FUNCTION_BLOCK FB_StationUnloadUc
VAR_INPUT
	Enable:				BOOL;
	System:				REFERENCE TO ST_System;
	Station:			REFERENCE TO ST_SystemStation;
	Error:				REFERENCE TO ST_Error;
	Setting:			REFERENCE TO ST_Setting;
	Recipe:				REFERENCE TO ST_Recipe;	
	Parameter:			REFERENCE TO ST_StationUnloadUc;
END_VAR
VAR_OUTPUT
END_VAR
VAR
	_i:					INT;
	_arrTon:		    ARRAY[0..20] OF TON;
	_arrFbErrorTag:		ARRAY[0..20] OF FB_ErrorTag;
	_arrState:			ARRAY[0..20] OF BOOL;
	_stHandshake: 		ST_StationUnloadUcHandshake;
END_VAR

A_Auto();
A_Home();

ACTION A_Auto:
CASE Station.iStepNow OF
	1000:
		Station.arrInfo[E_Language.Chinese]:="初始化完成 等待启动";
		IF Enable THEN
			Station.iStepNext:=1101;
		END_IF
	1101:
		Station.arrInfo[E_Language.Chinese]:="等待拆解站请求取料";
		IF Parameter.stHandshake.bRequestUc THEN
			Parameter.stHandshake.bResponseDismantling_Uc:=TRUE;
			Station.iStepNext:=1201;
		END_IF
	1201:
		Station.arrInfo[E_Language.Chinese]:="旋转气缸至取料位";
		IF Parameter.fbRotate.M_HomeRequest() THEN
			Station.iStepNext:=1251;
		END_IF
	1251:
		Station.arrInfo[E_Language.Chinese]:="升降气缸下降";
		IF  Parameter.fbLift.M_HomeRequest() THEN
			Station.iStepNext:=1301;
		END_IF
	1301:
		Station.arrInfo[E_Language.Chinese]:="夹紧气缸夹紧";
		IF Parameter.fbClamp.M_WorkRequest() THEN
			Station.iStepNext:=1401;
		END_IF
	1401:
		Station.arrInfo[E_Language.Chinese]:="升降气缸上升";
		IF Parameter.fbLift.M_WorkRequest() THEN
			Station.iStepNext:=1451;
		END_IF
	1451:
		Station.arrInfo[E_Language.Chinese]:="向下线体 请求放料";
		Parameter.stHandshake.bRequestUnloadLine:=TRUE;
		IF Parameter.stHandshake.bResponseUnladLine THEN
			Station.iStepNext:=1501;
		END_IF
	1501:
		Station.arrInfo[E_Language.Chinese]:="旋转气缸动作";
		IF Parameter.fbRotate.M_WorkRequest() THEN
			Station.iStepNext:=1551;
		END_IF
	1551:
		Station.arrInfo[E_Language.Chinese]:="等待复位取料请求";
		IF NOT Parameter.stHandshake.bRequestUc THEN
			Parameter.stHandshake.bResponseDismantling_Uc:=FALSE;
			Station.iStepNext:=1601;
		END_IF
	1601:
		Station.arrInfo[E_Language.Chinese]:="夹紧气缸松开";
		IF Parameter.fbClamp.M_HomeRequest() THEN
			Station.iStepNext:=1801;
		END_IF
	1801:
		Station.arrInfo[E_Language.Chinese]:="复位放料请求";
		Parameter.stHandshake.bRequestUnloadLine:=FALSE;
		IF NOT Parameter.stHandshake.bResponseUnladLine THEN
			Station.iStepNext:=1101;
		END_IF
END_CASE
END_ACTION

ACTION A_Home:
CASE Station.iStepNow OF
	0:
		Station.arrInfo[E_Language.Chinese]:="等待初始化";
		Parameter.stHandshake:=_stHandshake;
		Station.iStepNext:=SEL(Enable,1000,200);
	200:
		Station.arrInfo[E_Language.Chinese]:="升降气缸上升";
		IF Parameter.fbLift.M_WorkRequest() THEN
			Station.iStepNext:=300;
		END_IF
	300:
		Station.arrInfo[E_Language.Chinese]:="旋转气缸至下UC位";
		IF Parameter.fbRotate.M_WorkRequest() THEN
			Station.iStepNext:=400;
		END_IF
	400:
		Station.arrInfo[E_Language.Chinese]:="夹紧气缸复位";
		IF  Parameter.fbClamp.M_HomeRequest() THEN
			Station.iStepNext:=1000;
		END_IF
END_CASE
END_ACTION

END_FUNCTION_BLOCK

(* stored: Version 1.1.0.1, ProductVersion 3.1.4024.3
   POU FB_StationUnloadUc: Id {dcbe9bfd-225c-40dc-b3fa-9b9a7e2d07df}, SpecialFunc None
   Action A_Auto: Id {07211073-19ed-4810-8b75-27cce09f14a2}
   Action A_Home: Id {81728a20-c52b-4686-af61-ac93b7479c57} *)
